Staubli VAL3: iRack2.pgx

public program iRack2(num& nNum[] (dimensions=1))
begin
  nNum=dioGet(iRack2)
end
